{attribute 'GeneratedUsingTerminal: EP9214-0023-0019'}
{attribute addProperty BoxType "EP9214-0023-0019"}
{attribute addProperty Id "Enable_Control_Via_FieldbusAT %Q*BOOL1Global_ResetAT %Q*BOOL1"}
{attribute addProperty CRC "3061031735"}
{attribute addProperty Size "2"}
TYPE DPO_Outputs_Device_B673A337 EXTENDS OutputBase_10CEE7DE :
STRUCT
	{attribute addProperty Name "Enable_Control_Via_Fieldbus"}
	Enable_Control_Via_Fieldbus AT %Q* : BOOL;
	{attribute addProperty Name "Global_Reset"}
	Global_Reset AT %Q* : BOOL;
END_STRUCT
END_TYPE

(* stored: Version 1.2.0.0, ProductVersion 3.1.4024.11
   DUT DPO_Outputs_Device_B673A337: Id {7abf4bc2-0e52-471b-bbb6-67a89fb107eb} *)
